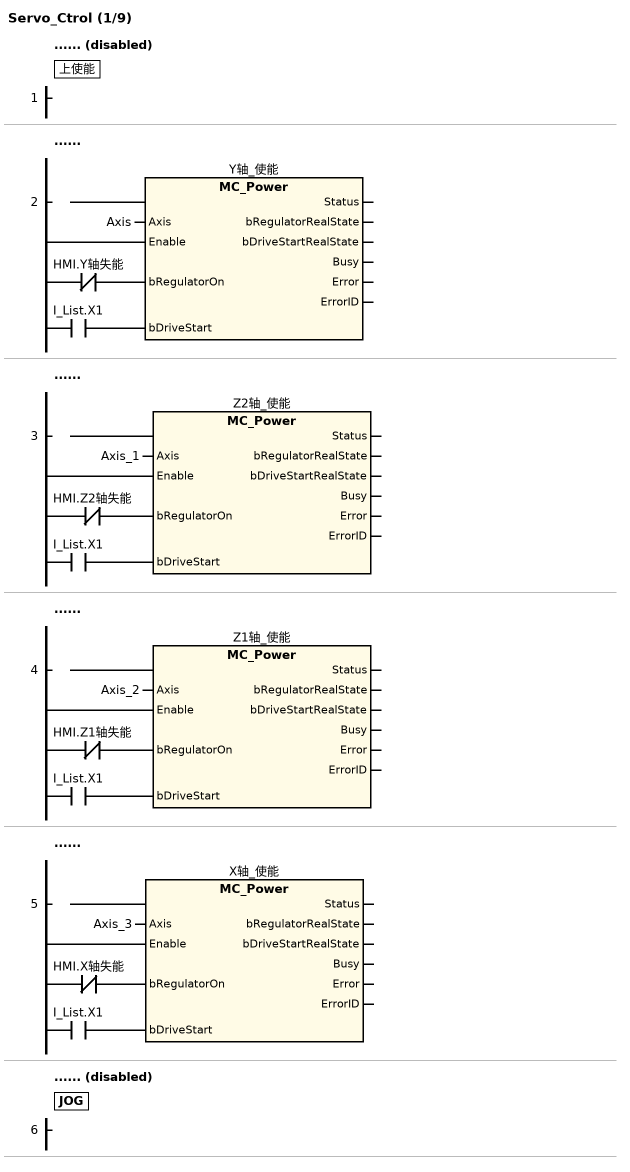
// NETWORK 1: ...... (disabled)
// label: 上使能

// NETWORK 2: ......
Y轴_使能(Axis := Axis, Enable := TRUE, bRegulatorOn := NOT HMI.Y轴失能, bDriveStart := I_List.X1); // MC_Power

// NETWORK 3: ......
Z2轴_使能(Axis := Axis_1, Enable := TRUE, bRegulatorOn := NOT HMI.Z2轴失能, bDriveStart := I_List.X1); // MC_Power

// NETWORK 4: ......
Z1轴_使能(Axis := Axis_2, Enable := TRUE, bRegulatorOn := NOT HMI.Z1轴失能, bDriveStart := I_List.X1); // MC_Power

// NETWORK 5: ......
X轴_使能(Axis := Axis_3, Enable := TRUE, bRegulatorOn := NOT HMI.X轴失能, bDriveStart := I_List.X1); // MC_Power

// NETWORK 6: ...... (disabled)
// label: JOG

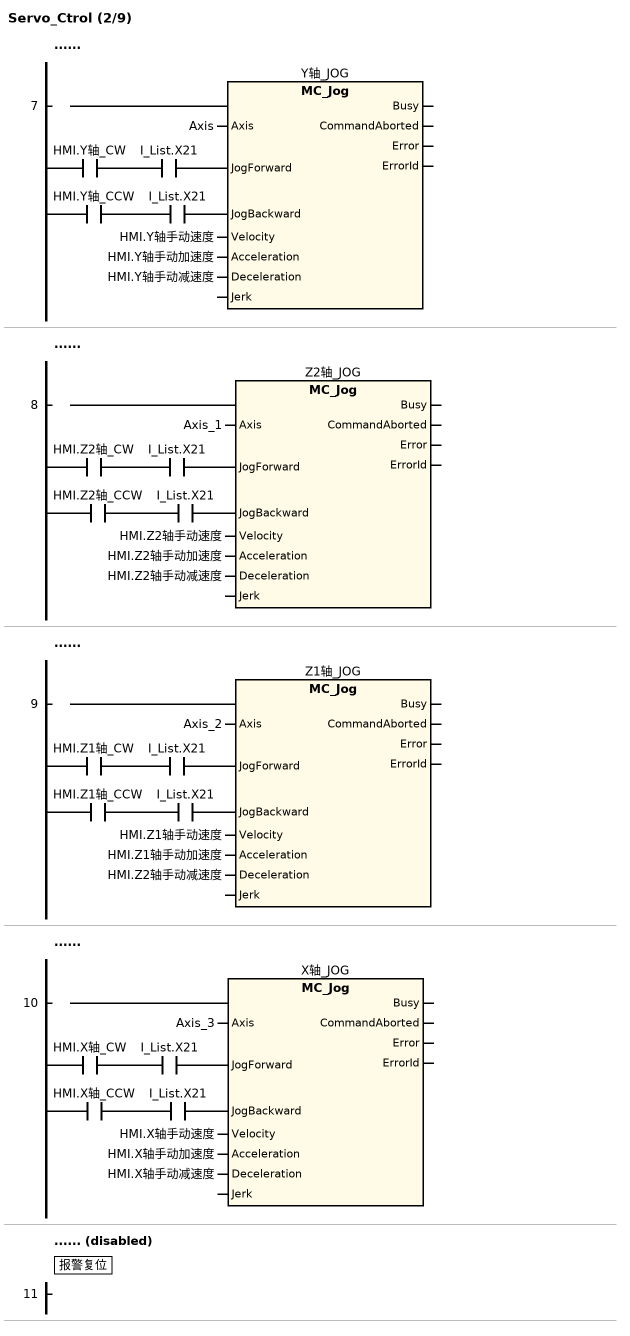
// NETWORK 7: ......
Y轴_JOG(
    Axis := Axis,
    JogForward := HMI.Y轴_CW AND I_List.X21,
    JogBackward := HMI.Y轴_CCW AND I_List.X21,
    Velocity := HMI.Y轴手动速度,
    Acceleration := HMI.Y轴手动加速度,
    Deceleration := HMI.Y轴手动减速度); // MC_Jog

// NETWORK 8: ......
Z2轴_JOG(
    Axis := Axis_1,
    JogForward := HMI.Z2轴_CW AND I_List.X21,
    JogBackward := HMI.Z2轴_CCW AND I_List.X21,
    Velocity := HMI.Z2轴手动速度,
    Acceleration := HMI.Z2轴手动加速度,
    Deceleration := HMI.Z2轴手动减速度); // MC_Jog

// NETWORK 9: ......
Z1轴_JOG(
    Axis := Axis_2,
    JogForward := HMI.Z1轴_CW AND I_List.X21,
    JogBackward := HMI.Z1轴_CCW AND I_List.X21,
    Velocity := HMI.Z1轴手动速度,
    Acceleration := HMI.Z1轴手动加速度,
    Deceleration := HMI.Z2轴手动减速度); // MC_Jog

// NETWORK 10: ......
X轴_JOG(
    Axis := Axis_3,
    JogForward := HMI.X轴_CW AND I_List.X21,
    JogBackward := HMI.X轴_CCW AND I_List.X21,
    Velocity := HMI.X轴手动速度,
    Acceleration := HMI.X轴手动加速度,
    Deceleration := HMI.X轴手动减速度); // MC_Jog

// NETWORK 11: ...... (disabled)
// label: 报警复位

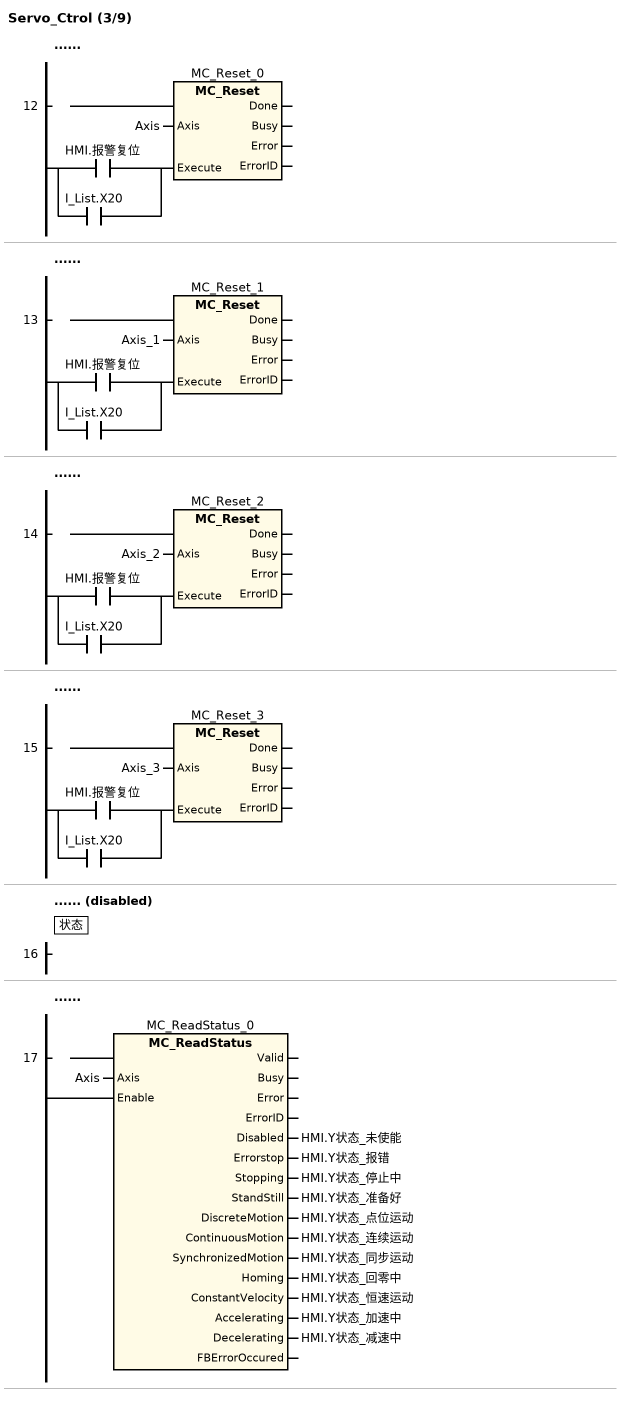
// NETWORK 12: ......
MC_Reset_0(Axis := Axis, Execute := HMI.报警复位 OR I_List.X20); // MC_Reset

// NETWORK 13: ......
MC_Reset_1(Axis := Axis_1, Execute := HMI.报警复位 OR I_List.X20); // MC_Reset

// NETWORK 14: ......
MC_Reset_2(Axis := Axis_2, Execute := HMI.报警复位 OR I_List.X20); // MC_Reset

// NETWORK 15: ......
MC_Reset_3(Axis := Axis_3, Execute := HMI.报警复位 OR I_List.X20); // MC_Reset

// NETWORK 16: ...... (disabled)
// label: 状态

// NETWORK 17: ......
MC_ReadStatus_0(
    Axis := Axis,
    Enable := TRUE,
    Disabled => HMI.Y状态_未使能,
    Errorstop => HMI.Y状态_报错,
    Stopping => HMI.Y状态_停止中,
    StandStill => HMI.Y状态_准备好,
    DiscreteMotion => HMI.Y状态_点位运动,
    ContinuousMotion => HMI.Y状态_连续运动,
    SynchronizedMotion => HMI.Y状态_同步运动,
    Homing => HMI.Y状态_回零中,
    ConstantVelocity => HMI.Y状态_恒速运动,
    Accelerating => HMI.Y状态_加速中,
    Decelerating => HMI.Y状态_减速中); // MC_ReadStatus

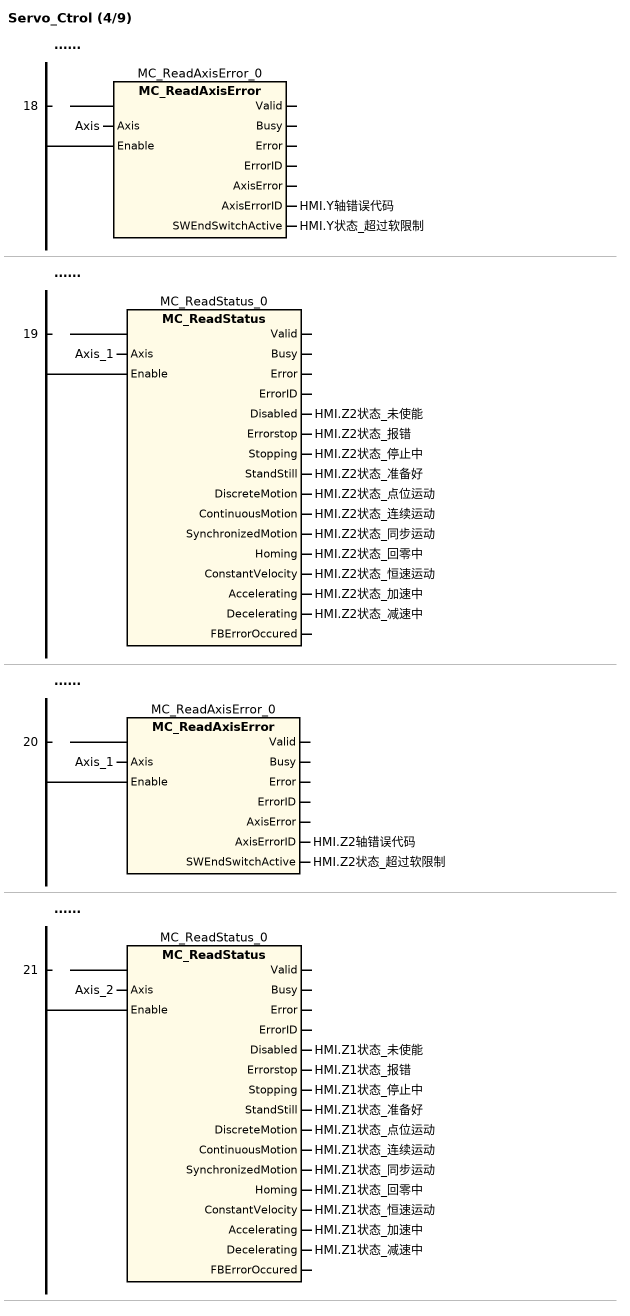
// NETWORK 18: ......
MC_ReadAxisError_0(
    Axis := Axis,
    Enable := TRUE,
    AxisErrorID => HMI.Y轴错误代码,
    SWEndSwitchActive => HMI.Y状态_超过软限制); // MC_ReadAxisError

// NETWORK 19: ......
MC_ReadStatus_0(
    Axis := Axis_1,
    Enable := TRUE,
    Disabled => HMI.Z2状态_未使能,
    Errorstop => HMI.Z2状态_报错,
    Stopping => HMI.Z2状态_停止中,
    StandStill => HMI.Z2状态_准备好,
    DiscreteMotion => HMI.Z2状态_点位运动,
    ContinuousMotion => HMI.Z2状态_连续运动,
    SynchronizedMotion => HMI.Z2状态_同步运动,
    Homing => HMI.Z2状态_回零中,
    ConstantVelocity => HMI.Z2状态_恒速运动,
    Accelerating => HMI.Z2状态_加速中,
    Decelerating => HMI.Z2状态_减速中); // MC_ReadStatus

// NETWORK 20: ......
MC_ReadAxisError_0(
    Axis := Axis_1,
    Enable := TRUE,
    AxisErrorID => HMI.Z2轴错误代码,
    SWEndSwitchActive => HMI.Z2状态_超过软限制); // MC_ReadAxisError

// NETWORK 21: ......
MC_ReadStatus_0(
    Axis := Axis_2,
    Enable := TRUE,
    Disabled => HMI.Z1状态_未使能,
    Errorstop => HMI.Z1状态_报错,
    Stopping => HMI.Z1状态_停止中,
    StandStill => HMI.Z1状态_准备好,
    DiscreteMotion => HMI.Z1状态_点位运动,
    ContinuousMotion => HMI.Z1状态_连续运动,
    SynchronizedMotion => HMI.Z1状态_同步运动,
    Homing => HMI.Z1状态_回零中,
    ConstantVelocity => HMI.Z1状态_恒速运动,
    Accelerating => HMI.Z1状态_加速中,
    Decelerating => HMI.Z1状态_减速中); // MC_ReadStatus

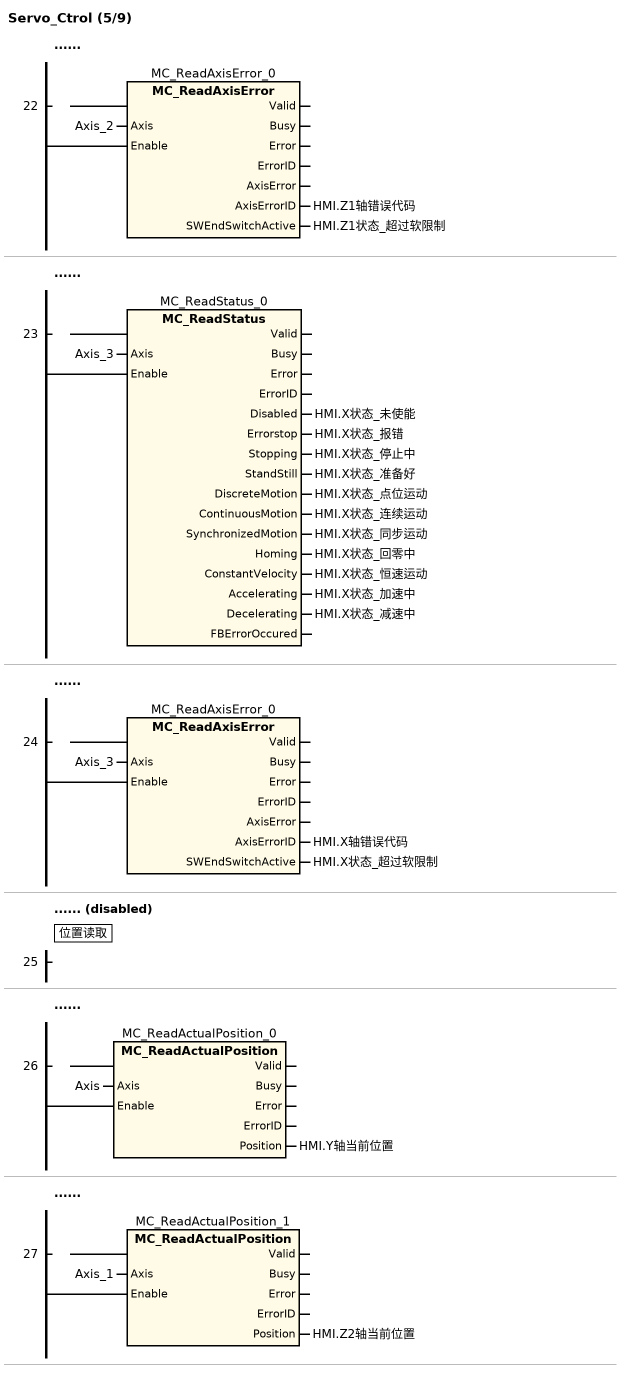
// NETWORK 22: ......
MC_ReadAxisError_0(
    Axis := Axis_2,
    Enable := TRUE,
    AxisErrorID => HMI.Z1轴错误代码,
    SWEndSwitchActive => HMI.Z1状态_超过软限制); // MC_ReadAxisError

// NETWORK 23: ......
MC_ReadStatus_0(
    Axis := Axis_3,
    Enable := TRUE,
    Disabled => HMI.X状态_未使能,
    Errorstop => HMI.X状态_报错,
    Stopping => HMI.X状态_停止中,
    StandStill => HMI.X状态_准备好,
    DiscreteMotion => HMI.X状态_点位运动,
    ContinuousMotion => HMI.X状态_连续运动,
    SynchronizedMotion => HMI.X状态_同步运动,
    Homing => HMI.X状态_回零中,
    ConstantVelocity => HMI.X状态_恒速运动,
    Accelerating => HMI.X状态_加速中,
    Decelerating => HMI.X状态_减速中); // MC_ReadStatus

// NETWORK 24: ......
MC_ReadAxisError_0(
    Axis := Axis_3,
    Enable := TRUE,
    AxisErrorID => HMI.X轴错误代码,
    SWEndSwitchActive => HMI.X状态_超过软限制); // MC_ReadAxisError

// NETWORK 25: ...... (disabled)
// label: 位置读取

// NETWORK 26: ......
MC_ReadActualPosition_0(Axis := Axis, Enable := TRUE, Position => HMI.Y轴当前位置); // MC_ReadActualPosition

// NETWORK 27: ......
MC_ReadActualPosition_1(Axis := Axis_1, Enable := TRUE, Position => HMI.Z2轴当前位置); // MC_ReadActualPosition

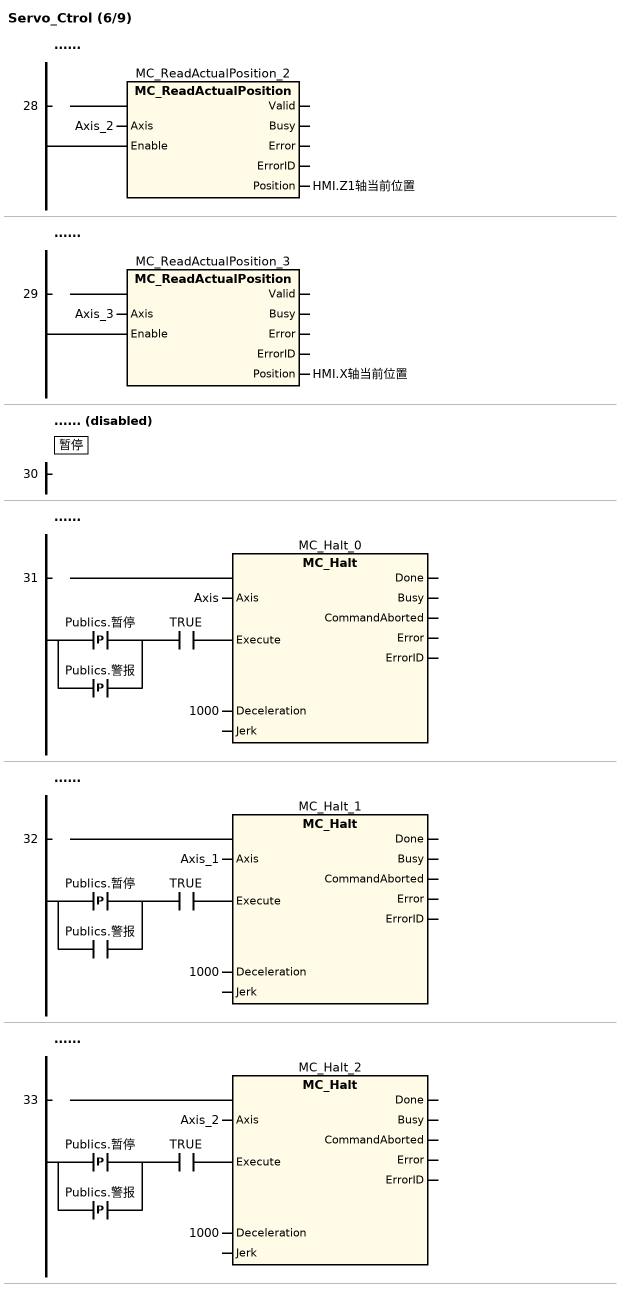
// NETWORK 28: ......
MC_ReadActualPosition_2(Axis := Axis_2, Enable := TRUE, Position => HMI.Z1轴当前位置); // MC_ReadActualPosition

// NETWORK 29: ......
MC_ReadActualPosition_3(Axis := Axis_3, Enable := TRUE, Position => HMI.X轴当前位置); // MC_ReadActualPosition

// NETWORK 30: ...... (disabled)
// label: 暂停

// NETWORK 31: ......
_rt1(CLK := Publics.暂停);
_rt2(CLK := Publics.警报);
MC_Halt_0(Axis := Axis, Execute := (_rt1.Q OR _rt2.Q) AND TRUE, Deceleration := 1000); // MC_Halt

// NETWORK 32: ......
_rt3(CLK := Publics.暂停);
MC_Halt_1(Axis := Axis_1, Execute := (_rt3.Q OR Publics.警报) AND TRUE, Deceleration := 1000); // MC_Halt

// NETWORK 33: ......
_rt4(CLK := Publics.暂停);
_rt5(CLK := Publics.警报);
MC_Halt_2(Axis := Axis_2, Execute := (_rt4.Q OR _rt5.Q) AND TRUE, Deceleration := 1000); // MC_Halt

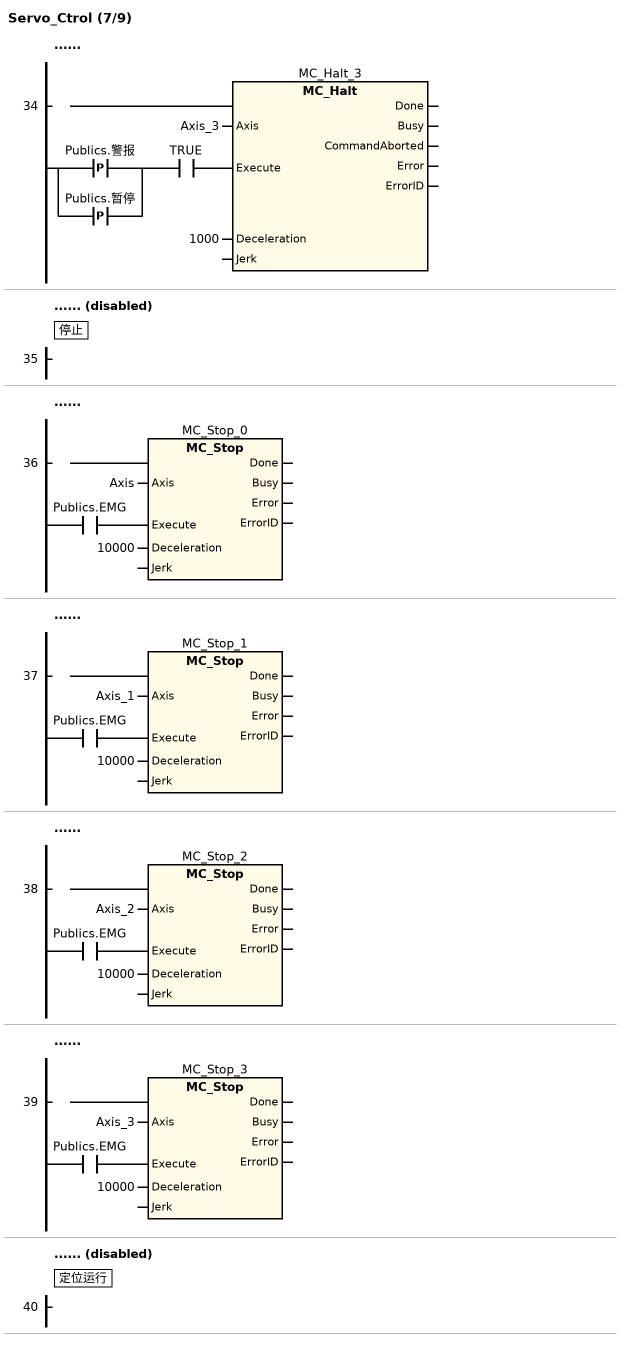
// NETWORK 34: ......
_rt6(CLK := Publics.警报);
_rt7(CLK := Publics.暂停);
MC_Halt_3(Axis := Axis_3, Execute := (_rt6.Q OR _rt7.Q) AND TRUE, Deceleration := 1000); // MC_Halt

// NETWORK 35: ...... (disabled)
// label: 停止

// NETWORK 36: ......
MC_Stop_0(Axis := Axis, Execute := Publics.EMG, Deceleration := 10000); // MC_Stop

// NETWORK 37: ......
MC_Stop_1(Axis := Axis_1, Execute := Publics.EMG, Deceleration := 10000); // MC_Stop

// NETWORK 38: ......
MC_Stop_2(Axis := Axis_2, Execute := Publics.EMG, Deceleration := 10000); // MC_Stop

// NETWORK 39: ......
MC_Stop_3(Axis := Axis_3, Execute := Publics.EMG, Deceleration := 10000); // MC_Stop

// NETWORK 40: ...... (disabled)
// label: 定位运行

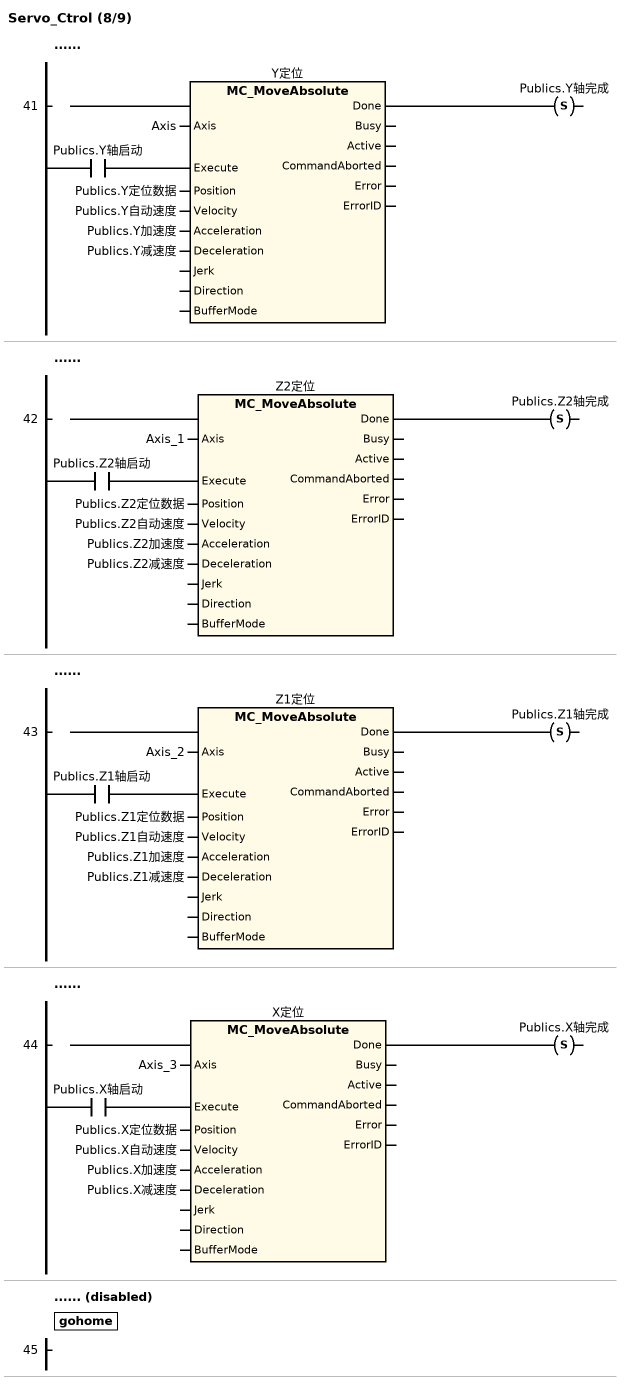
// NETWORK 41: ......
Y定位(
    Axis := Axis,
    Execute := Publics.Y轴启动,
    Position := Publics.Y定位数据,
    Velocity := Publics.Y自动速度,
    Acceleration := Publics.Y加速度,
    Deceleration := Publics.Y减速度); // MC_MoveAbsolute
Publics.Y轴完成 S= Y定位.Done;

// NETWORK 42: ......
Z2定位(
    Axis := Axis_1,
    Execute := Publics.Z2轴启动,
    Position := Publics.Z2定位数据,
    Velocity := Publics.Z2自动速度,
    Acceleration := Publics.Z2加速度,
    Deceleration := Publics.Z2减速度); // MC_MoveAbsolute
Publics.Z2轴完成 S= Z2定位.Done;

// NETWORK 43: ......
Z1定位(
    Axis := Axis_2,
    Execute := Publics.Z1轴启动,
    Position := Publics.Z1定位数据,
    Velocity := Publics.Z1自动速度,
    Acceleration := Publics.Z1加速度,
    Deceleration := Publics.Z1减速度); // MC_MoveAbsolute
Publics.Z1轴完成 S= Z1定位.Done;

// NETWORK 44: ......
X定位(
    Axis := Axis_3,
    Execute := Publics.X轴启动,
    Position := Publics.X定位数据,
    Velocity := Publics.X自动速度,
    Acceleration := Publics.X加速度,
    Deceleration := Publics.X减速度); // MC_MoveAbsolute
Publics.X轴完成 S= X定位.Done;

// NETWORK 45: ...... (disabled)
// label: gohome

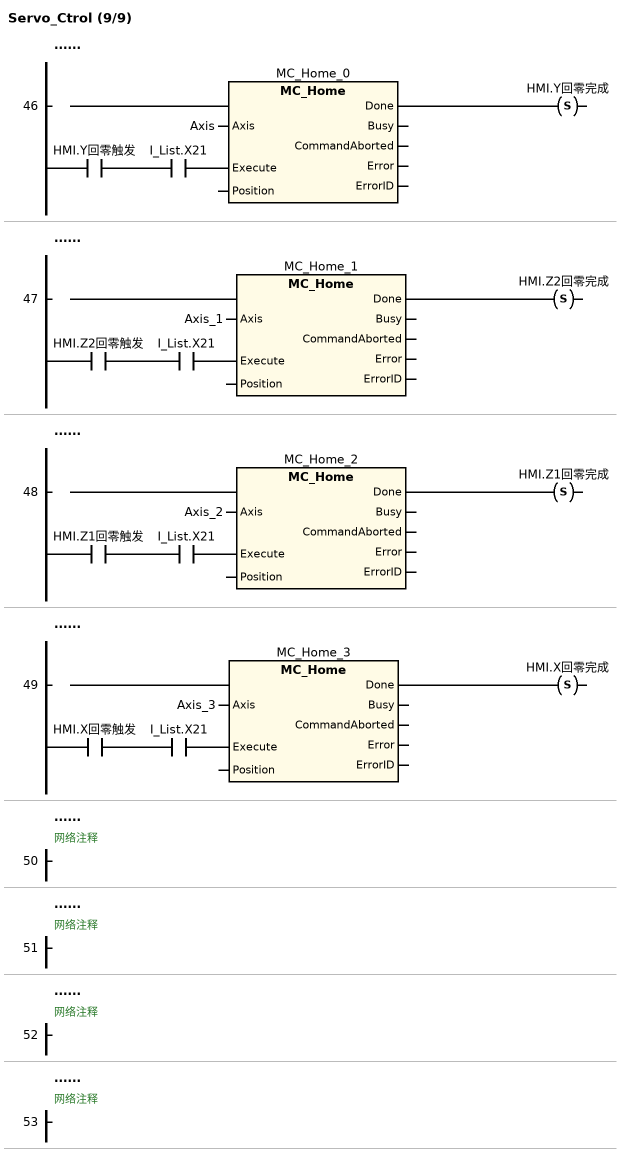
// NETWORK 46: ......
MC_Home_0(Axis := Axis, Execute := HMI.Y回零触发 AND I_List.X21); // MC_Home
HMI.Y回零完成 S= MC_Home_0.Done;

// NETWORK 47: ......
MC_Home_1(Axis := Axis_1, Execute := HMI.Z2回零触发 AND I_List.X21); // MC_Home
HMI.Z2回零完成 S= MC_Home_1.Done;

// NETWORK 48: ......
MC_Home_2(Axis := Axis_2, Execute := HMI.Z1回零触发 AND I_List.X21); // MC_Home
HMI.Z1回零完成 S= MC_Home_2.Done;

// NETWORK 49: ......
MC_Home_3(Axis := Axis_3, Execute := HMI.X回零触发 AND I_List.X21); // MC_Home
HMI.X回零完成 S= MC_Home_3.Done;

// NETWORK 50: ......
// 网络注释

// NETWORK 51: ......
// 网络注释

// NETWORK 52: ......
// 网络注释

// NETWORK 53: ......
// 网络注释

END_PROGRAM

// Device/Application/ITF
INTERFACE ITF

END_INTERFACE

// Device/Application/POU
PROGRAM POU
VAR
	当前步: uint;
	下一步: uint;
	定位位置: ARRAY[0..3] OF Lreal;
	LS_4AxisLine_0: LS_4AxisLine;
	避开扫描周期: BOOL;
	所有轴启动: BOOL;
	轴运行完成: BOOL;
END_VAR
VAR // added by the converter: edge detectors and wires of the graphical bodies
    _w1, _w2, _w3, _w4, _w5, _w6, _w7, _w8, _w9, _w10, _w11, _w12 : BOOL;
END_VAR

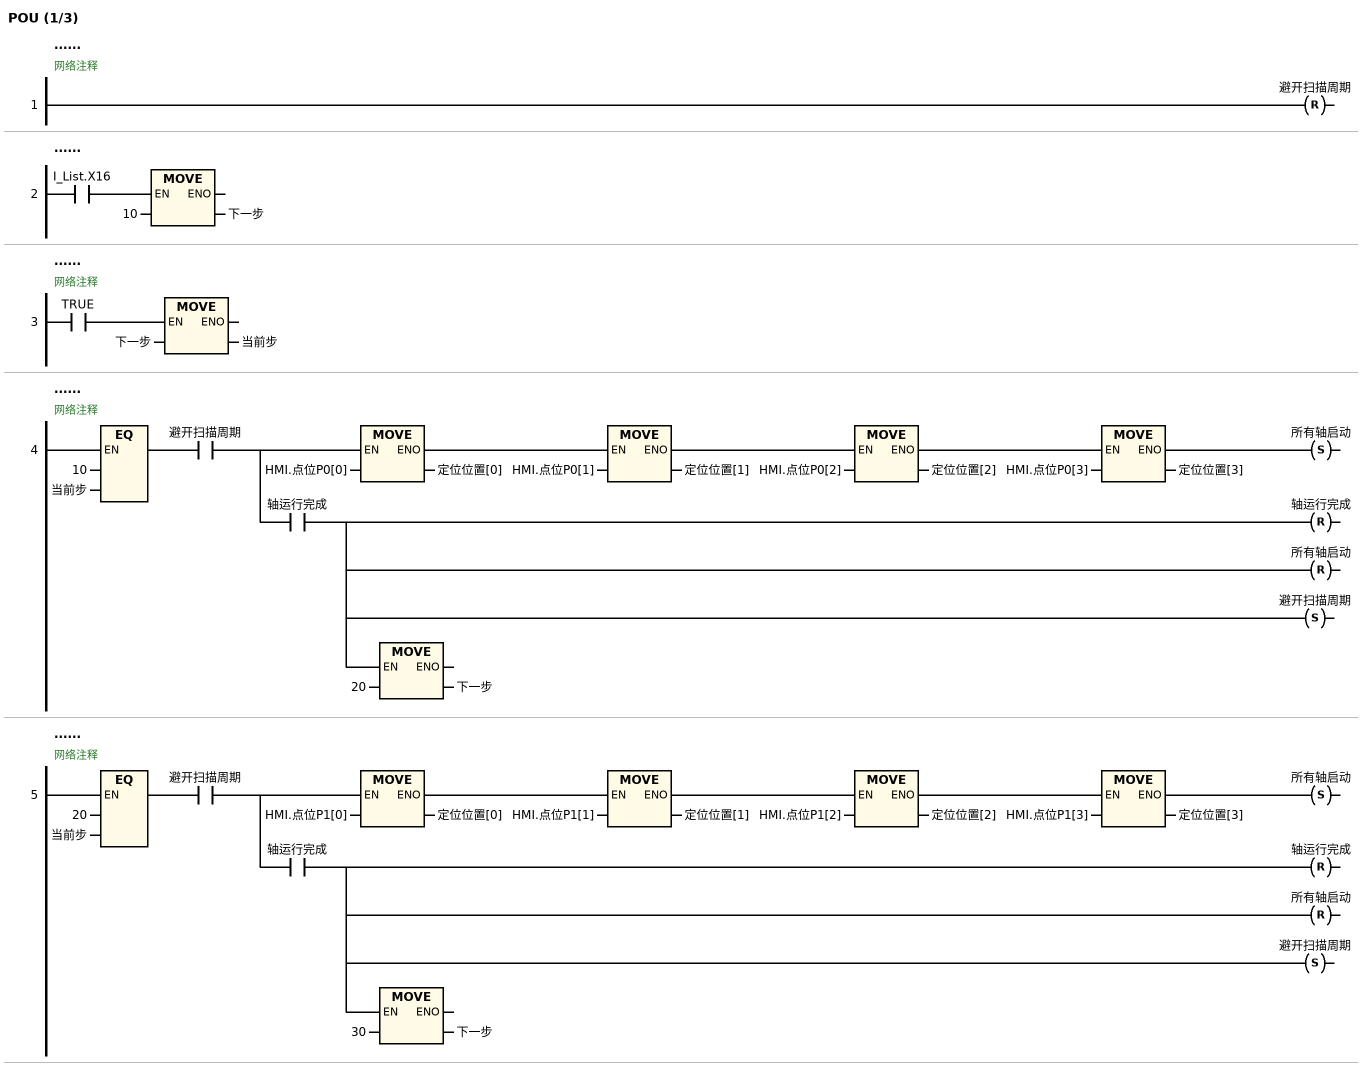
// NETWORK 1: ......
// 网络注释
避开扫描周期 R= TRUE;

// NETWORK 2: ......
IF I_List.X16 THEN 下一步 := 10; END_IF

// NETWORK 3: ......
// 网络注释
当前步 := 下一步;

// NETWORK 4: ......
// 网络注释
_w1 := 10 = 当前步 AND 避开扫描周期;
IF _w1 THEN 定位位置[0] := HMI.点位P0[0]; END_IF
IF _w1 THEN 定位位置[1] := HMI.点位P0[1]; END_IF
IF _w1 THEN 定位位置[2] := HMI.点位P0[2]; END_IF
IF _w1 THEN 定位位置[3] := HMI.点位P0[3]; END_IF
所有轴启动 S= _w1;
_w2 := _w1 AND 轴运行完成;
轴运行完成 R= _w2;
所有轴启动 R= _w2;
避开扫描周期 S= _w2;
IF _w2 THEN 下一步 := 20; END_IF

// NETWORK 5: ......
// 网络注释
_w3 := 20 = 当前步 AND 避开扫描周期;
IF _w3 THEN 定位位置[0] := HMI.点位P1[0]; END_IF
IF _w3 THEN 定位位置[1] := HMI.点位P1[1]; END_IF
IF _w3 THEN 定位位置[2] := HMI.点位P1[2]; END_IF
IF _w3 THEN 定位位置[3] := HMI.点位P1[3]; END_IF
所有轴启动 S= _w3;
_w4 := _w3 AND 轴运行完成;
轴运行完成 R= _w4;
所有轴启动 R= _w4;
避开扫描周期 S= _w4;
IF _w4 THEN 下一步 := 30; END_IF

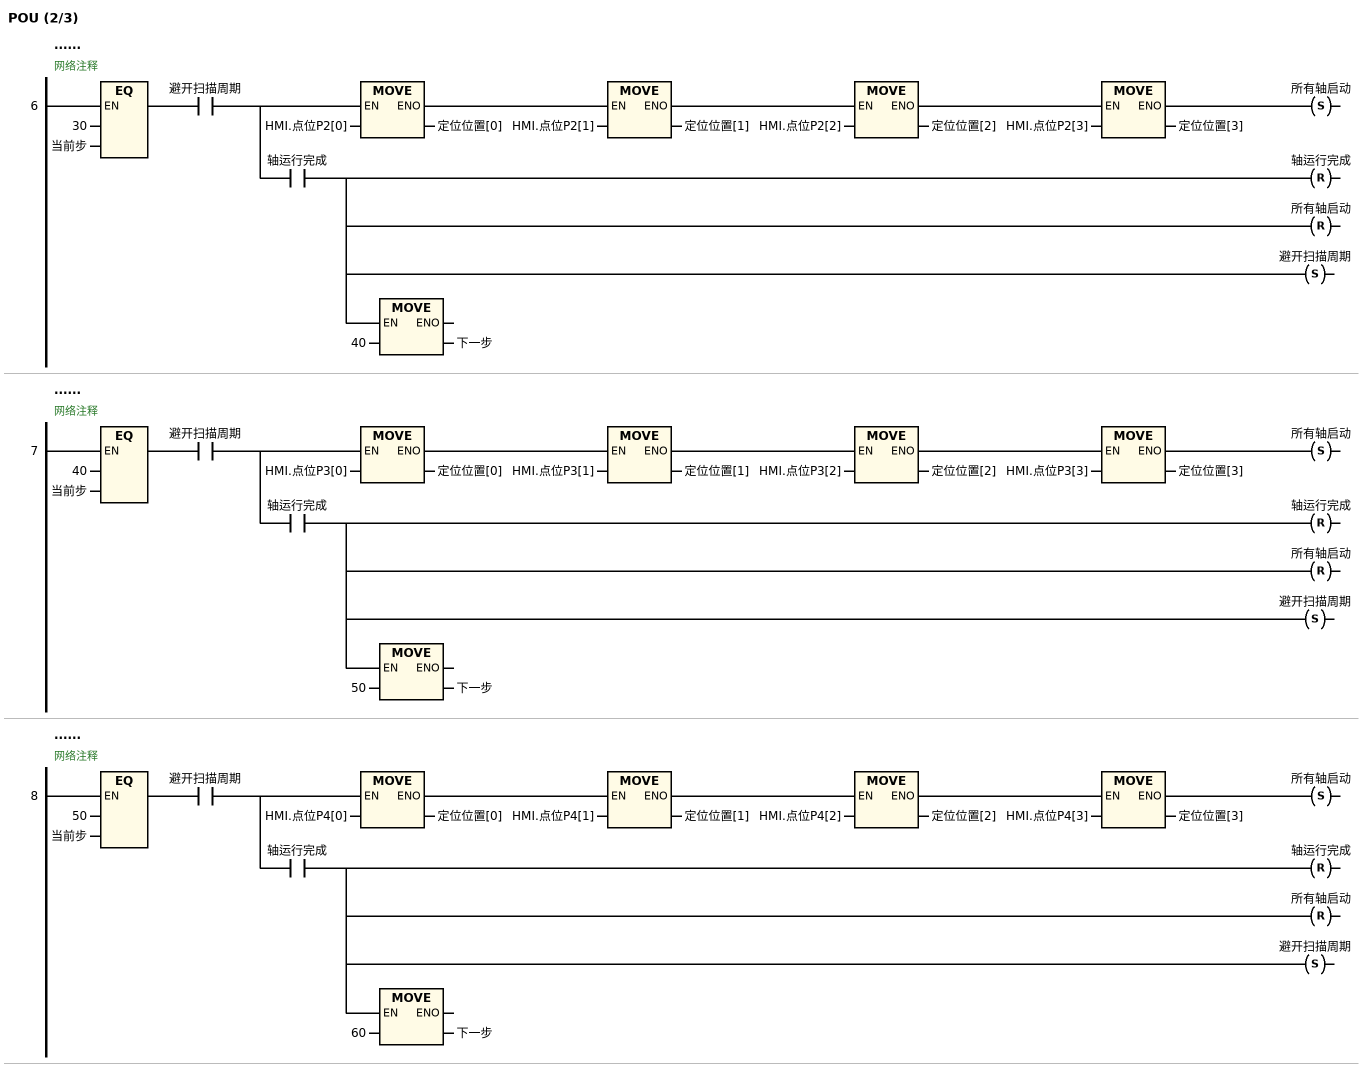
// NETWORK 6: ......
// 网络注释
_w5 := 30 = 当前步 AND 避开扫描周期;
IF _w5 THEN 定位位置[0] := HMI.点位P2[0]; END_IF
IF _w5 THEN 定位位置[1] := HMI.点位P2[1]; END_IF
IF _w5 THEN 定位位置[2] := HMI.点位P2[2]; END_IF
IF _w5 THEN 定位位置[3] := HMI.点位P2[3]; END_IF
所有轴启动 S= _w5;
_w6 := _w5 AND 轴运行完成;
轴运行完成 R= _w6;
所有轴启动 R= _w6;
避开扫描周期 S= _w6;
IF _w6 THEN 下一步 := 40; END_IF

// NETWORK 7: ......
// 网络注释
_w7 := 40 = 当前步 AND 避开扫描周期;
IF _w7 THEN 定位位置[0] := HMI.点位P3[0]; END_IF
IF _w7 THEN 定位位置[1] := HMI.点位P3[1]; END_IF
IF _w7 THEN 定位位置[2] := HMI.点位P3[2]; END_IF
IF _w7 THEN 定位位置[3] := HMI.点位P3[3]; END_IF
所有轴启动 S= _w7;
_w8 := _w7 AND 轴运行完成;
轴运行完成 R= _w8;
所有轴启动 R= _w8;
避开扫描周期 S= _w8;
IF _w8 THEN 下一步 := 50; END_IF

// NETWORK 8: ......
// 网络注释
_w9 := 50 = 当前步 AND 避开扫描周期;
IF _w9 THEN 定位位置[0] := HMI.点位P4[0]; END_IF
IF _w9 THEN 定位位置[1] := HMI.点位P4[1]; END_IF
IF _w9 THEN 定位位置[2] := HMI.点位P4[2]; END_IF
IF _w9 THEN 定位位置[3] := HMI.点位P4[3]; END_IF
所有轴启动 S= _w9;
_w10 := _w9 AND 轴运行完成;
轴运行完成 R= _w10;
所有轴启动 R= _w10;
避开扫描周期 S= _w10;
IF _w10 THEN 下一步 := 60; END_IF

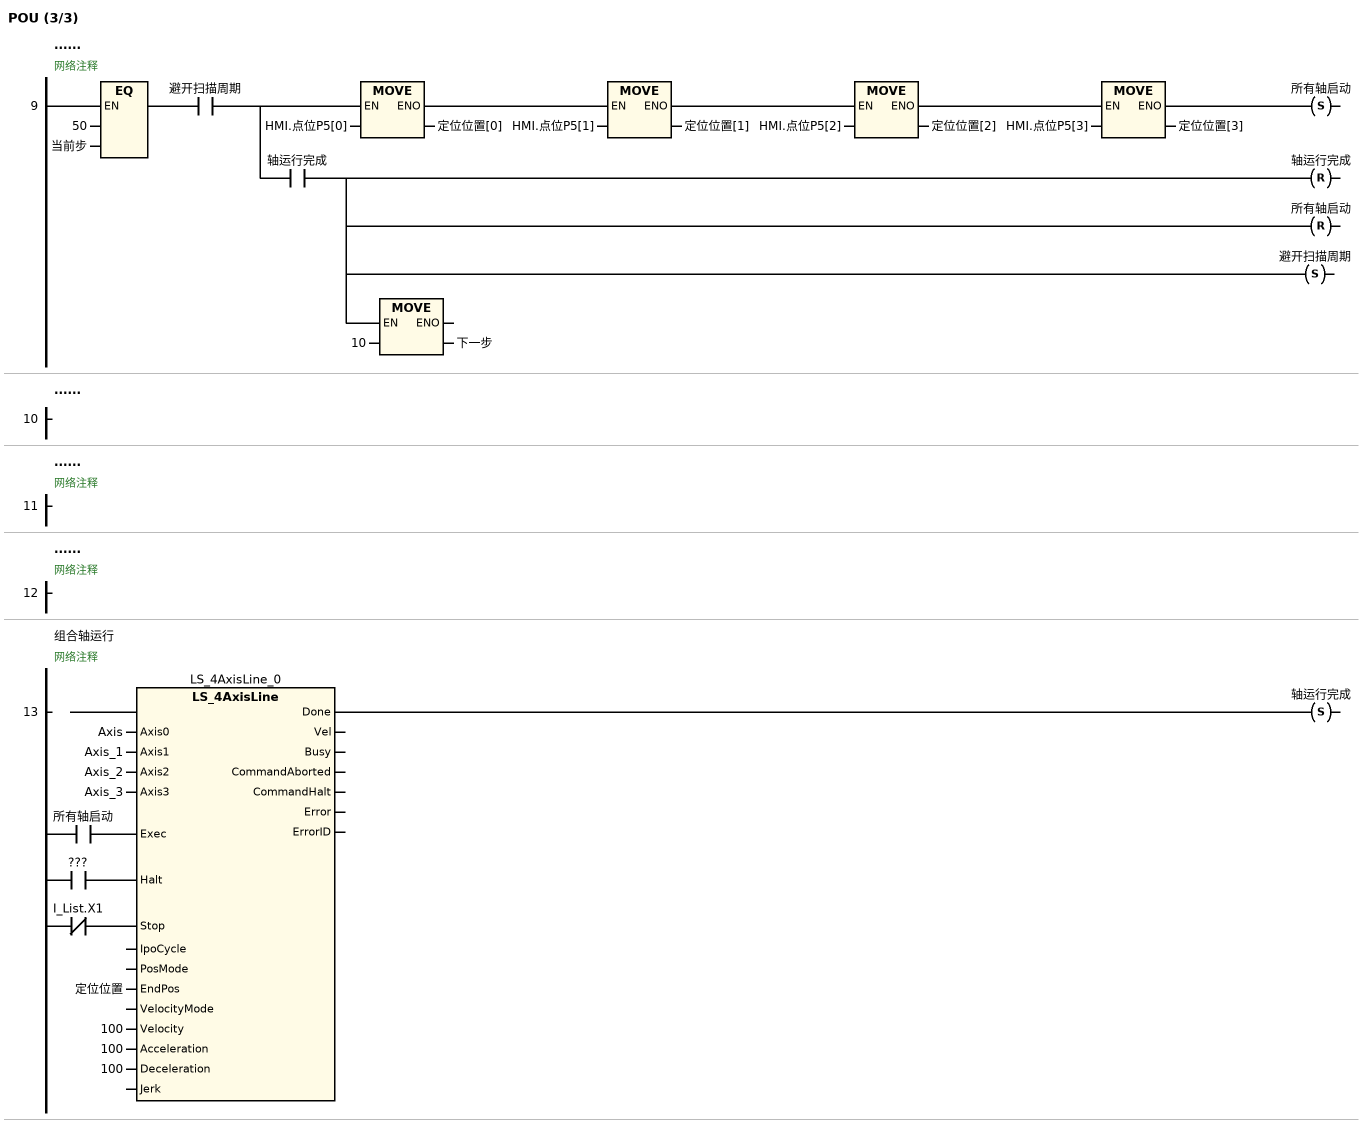
// NETWORK 9: ......
// 网络注释
_w11 := 50 = 当前步 AND 避开扫描周期;
IF _w11 THEN 定位位置[0] := HMI.点位P5[0]; END_IF
IF _w11 THEN 定位位置[1] := HMI.点位P5[1]; END_IF
IF _w11 THEN 定位位置[2] := HMI.点位P5[2]; END_IF
IF _w11 THEN 定位位置[3] := HMI.点位P5[3]; END_IF
所有轴启动 S= _w11;
_w12 := _w11 AND 轴运行完成;
轴运行完成 R= _w12;
所有轴启动 R= _w12;
避开扫描周期 S= _w12;
IF _w12 THEN 下一步 := 10; END_IF

// NETWORK 10: ......

// NETWORK 11: ......
// 网络注释

// NETWORK 12: ......
// 网络注释

// NETWORK 13: 组合轴运行
// 网络注释
LS_4AxisLine_0(
    Axis0 := Axis,
    Axis1 := Axis_1,
    Axis2 := Axis_2,
    Axis3 := Axis_3,
    Exec := 所有轴启动,
    Stop := NOT I_List.X1,
    EndPos := 定位位置,
    Velocity := 100,
    Acceleration := 100,
    Deceleration := 100); // LS_4AxisLine
轴运行完成 S= LS_4AxisLine_0.Done;

END_PROGRAM

// Device/Application/Visualization
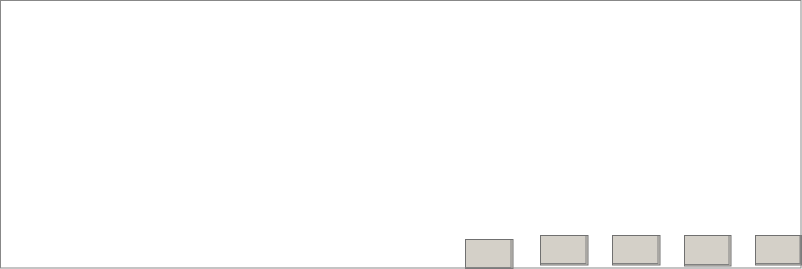
VISUALIZATION Visualization  // 802x269
    Button (465,239 48x30)
        toggle POU_1.M0
    Button (540,235 48x30)
        tap POU_1.M1
    Button (612,235 48x30)
        tap POU_1.M2
    Button (684,235 47x31)
        toggle POU_1.M3
    Button (755,235 47x30)
        tap POU_1.M4
END_VISUALIZATION
